// TIA Portal V19 export
FUNCTION_BLOCK "TYPIC_C103_IF_HVN"   // FB18, FBD
TITLE = TYPIC_C103_IF_HVN: ALSB NB
{ S7_Optimized_Access := 'TRUE' }
AUTHOR : OCOTECH
FAMILY : Typical
NAME : C103.702
// Logisch Object Besturing: C103.803
// 
// De interne functie laagspanningsverdeelbord no break verzorgt de bewaking van een laagspanningsverdeelbord no break.
// stored: MemoryReserve 10, SetENOAutomatically false
   VAR_INPUT
      EXT_AUT { ExternalAccessible := 'False'; ExternalVisible := 'False'; ExternalWritable := 'False'} : Bool;   // Externe (hoofd) beveiliging (1 = OK)
      EXT_HW { ExternalAccessible := 'False'; ExternalVisible := 'False'; ExternalWritable := 'False'} : Bool;   // Sturings hardware (PLC) bewaking (1 = OK)
      IN_PWR1 { ExternalAccessible := 'False'; ExternalVisible := 'False'; ExternalWritable := 'False'} : Real;   // Actief vermogen
      IN_PWR2 { ExternalAccessible := 'False'; ExternalVisible := 'False'; ExternalWritable := 'False'} : Real;   // Reactief vermogen
      IN_SPA_1 { ExternalAccessible := 'False'; ExternalVisible := 'False'; ExternalWritable := 'False'} : Real;   // Spanningsniveau lijn 1
      IN_SPA_2 { ExternalAccessible := 'False'; ExternalVisible := 'False'; ExternalWritable := 'False'} : Real;   // Spanningsniveau lijn 2
      IN_SPA_3 { ExternalAccessible := 'False'; ExternalVisible := 'False'; ExternalWritable := 'False'} : Real;   // Spanningsniveau lijn 3
      IN_SPA_4 { ExternalAccessible := 'False'; ExternalVisible := 'False'; ExternalWritable := 'False'} : Real;   // Lijnspanning L1-L2
      IN_SPA_5 { ExternalAccessible := 'False'; ExternalVisible := 'False'; ExternalWritable := 'False'} : Real;   // Lijnspanning L2-L3
      IN_SPA_6 { ExternalAccessible := 'False'; ExternalVisible := 'False'; ExternalWritable := 'False'} : Real;   // Lijnspanning L1-L3
      IN_STR_1 { ExternalAccessible := 'False'; ExternalVisible := 'False'; ExternalWritable := 'False'} : Real;   // Stroom lijn 1
      IN_STR_2 { ExternalAccessible := 'False'; ExternalVisible := 'False'; ExternalWritable := 'False'} : Real;   // Stroom lijn 2
      IN_STR_3 { ExternalAccessible := 'False'; ExternalVisible := 'False'; ExternalWritable := 'False'} : Real;   // Stroom lijn 3
      IN_STR_4 { ExternalAccessible := 'False'; ExternalVisible := 'False'; ExternalWritable := 'False'} : Real;   // Stroom nulleider
      IN_PHI { ExternalAccessible := 'False'; ExternalVisible := 'False'; ExternalWritable := 'False'} : Real;   // Arbeidsfactor
      IN_AUT_TOE { ExternalAccessible := 'False'; ExternalVisible := 'False'; ExternalWritable := 'False'} : Bool;   // Standmelding van elke vermogenschakelaar TOE [gesloten]
      IN_SCL1 { ExternalAccessible := 'False'; ExternalVisible := 'False'; ExternalWritable := 'False'} : Bool;   // Standmelding externe bypass netspanning
      IN_SCL2 { ExternalAccessible := 'False'; ExternalVisible := 'False'; ExternalWritable := 'False'} : Bool;   // Standmelding aankomstschakelaar UPS
   END_VAR
   VAR_OUTPUT
      VAR_IF_HVN { ExternalAccessible := 'False'; ExternalVisible := 'False'; ExternalWritable := 'False'} : "C103_VAR_IF_HVN_TYPIC";   // Struct met alle variabelen naar bovenliggende functies
   END_VAR
   VAR
      STO { ExternalWritable := 'False'} : Struct   // Storingen
         A001 { ExternalAccessible := 'False'; ExternalVisible := 'False'} : Bool;   // Laagspanningsverdeelbord no break beveiliging aangesproken
         A002 { ExternalAccessible := 'False'; ExternalVisible := 'False'} : Bool;   // Laagspanningsverdeelbord no break in storing
      END_STRUCT;
      VAR { ExternalWritable := 'False'} : Struct   // Variabelen
         PWR1 { ExternalAccessible := 'False'; ExternalVisible := 'False'} : Real;   // Actief vermogen
         PWR2 { ExternalAccessible := 'False'; ExternalVisible := 'False'} : Real;   // Reactief vermogen
         SPA_1 { ExternalAccessible := 'False'; ExternalVisible := 'False'} : Real;   // Spanningsniveau lijn 1
         SPA_2 { ExternalAccessible := 'False'; ExternalVisible := 'False'} : Real;   // Spanningsniveau lijn 2
         SPA_3 { ExternalAccessible := 'False'; ExternalVisible := 'False'} : Real;   // Spanningsniveau lijn 3
         SPA_4 { ExternalAccessible := 'False'; ExternalVisible := 'False'} : Real;   // Lijnspanning L1-L2
         SPA_5 { ExternalAccessible := 'False'; ExternalVisible := 'False'} : Real;   // Lijnspanning L2-L3
         SPA_6 { ExternalAccessible := 'False'; ExternalVisible := 'False'} : Real;   // Lijnspanning L1-L3
         STR_1 { ExternalAccessible := 'False'; ExternalVisible := 'False'} : Real;   // Stroom lijn 1
         STR_2 { ExternalAccessible := 'False'; ExternalVisible := 'False'} : Real;   // Stroom lijn 2
         STR_3 { ExternalAccessible := 'False'; ExternalVisible := 'False'} : Real;   // Stroom lijn 3
         STR_4 { ExternalAccessible := 'False'; ExternalVisible := 'False'} : Real;   // Stroom nulleider
         PHI { ExternalAccessible := 'False'; ExternalVisible := 'False'} : Real;   // Arbeidsfactor
         AUT_TOE { ExternalAccessible := 'False'; ExternalVisible := 'False'} : Bool;   // Standmelding van elke vermogenschakelaar TOE [gesloten]
         SCL1 { ExternalAccessible := 'False'; ExternalVisible := 'False'} : Bool;   // Standmelding externe bypass netspanning
         SCL2 { ExternalAccessible := 'False'; ExternalVisible := 'False'} : Bool;   // Standmelding aankomstschakelaar UPS
      END_STRUCT;
   END_VAR
BEGIN

REGION Network 1: START
END_REGION

REGION Network 2: +++ Verwerking meetwaarden en statussen +++
   // De meetwaarde en status wordt ontvangen vanuit de interne sturing.
END_REGION

REGION Network 3: +++ Storingen +++
   // Combinatie van de storingen
END_REGION

REGION Network 4: Storing A001: Laagspanningsverdeelbord no break beveiliging aangesproken
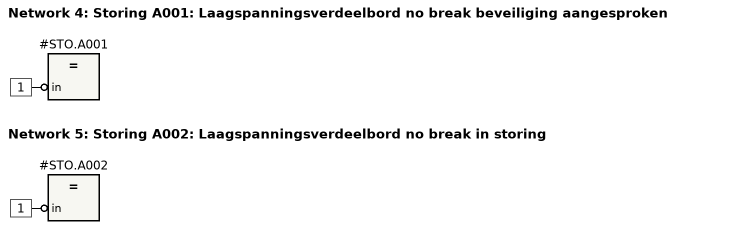
   #STO.A001 := NOT 1;
END_REGION

REGION Network 5: Storing A002: Laagspanningsverdeelbord no break in storing
   #STO.A002 := NOT 1;
END_REGION

REGION Network 6 (SCL): EINDE
   // Variabelen van intern scada rakvlak naar outputs copieren
   #VAR_IF_HVN.PWR1 := #VAR.PWR1;
   #VAR_IF_HVN.PWR2 := #VAR.PWR2;
   #VAR_IF_HVN.SPA_1 := #VAR.SPA_1;
   #VAR_IF_HVN.SPA_2 := #VAR.SPA_2;
   #VAR_IF_HVN.SPA_3 := #VAR.SPA_3;
   #VAR_IF_HVN.SPA_4 := #VAR.SPA_4;
   #VAR_IF_HVN.SPA_5 := #VAR.SPA_5;
   #VAR_IF_HVN.SPA_6 := #VAR.SPA_6;
   #VAR_IF_HVN.STR_1 := #VAR.STR_1;
   #VAR_IF_HVN.STR_2 := #VAR.STR_2;
   #VAR_IF_HVN.STR_3 := #VAR.STR_3;
   #VAR_IF_HVN.STR_4 := #VAR.STR_4;
   #VAR_IF_HVN.PHI := #VAR.PHI;
   #VAR_IF_HVN.AUT_TOE := #VAR.AUT_TOE;
   #VAR_IF_HVN.SCL1 := #VAR.SCL1;
   #VAR_IF_HVN.SCL2 := #VAR.SCL2;
END_REGION
END_FUNCTION_BLOCK
